{attribute 'qualified_only'}
{attribute 'strict'}
TYPE tStatiMSF :
(
	S0_Spento := 0,
	S1_RipristinoMandrino,
	S2_AttesaPezzo,
	S3_PausaIngresso,
	S4_Caricamento,
	S5_DiscesaMandrino,
	S6_SalitaMandrino,
	S7_Scarico,
	S8_PausaScarico,
	SE_Emergenza,
	SA1_RipristinoMAndrino,
	SA2_UscitaPezzo
);
END_TYPE

(* stored: Version 1.1.0.1, ProductVersion 3.1.4024.12
   EnumerationTextList tStatiMSF: Id {af65e22f-1c5f-4baa-8e2c-73f79ac36412} *)
